# B&R Automation Studio project DemoWall
Automation Studio 4.3.6.57 SP; technology packages: Acp10Arnc0 3.18.2, mapp 1.62.1

## Configuration HardwareConfig1

CPU X20CP1382, AutomationRuntime E4.34, Build 4.1.2, Vc V4.34.3, Safety 1.6

### Task classes (Cpu.sw)
```
Cyclic#1:
  AnalogInpu <- Sources.SimPanel.AnalogInputControl.AnalogInputControl.prg
  DigitalInp <- Sources.SimPanel.DigitalInputControl.DigitalInputControl.prg
  AnalogOutp <- Sources.SimPanel.AnalogOutputControl.AnalogOutputControl.prg
  DigitalOup <- Sources.SimPanel.DigitalOutputControl.DigitalOuputControl.prg
DataObjects: Acp10sys
NcDataObjects: acp10etxen <- DriveAxisConfig.AxisAdditionalFiles.acp10etxen.dob, gAxis01a <- DriveAxisConfig.ACOPOS_P3_3axis.gAxis01obj.gAxis01a.dob, gAxis01i <- DriveAxisConfig.ACOPOS_P3_3axis.gAxis01obj.gAxis01i.dob, gAxis02a <- DriveAxisConfig.ACOPOS_P3_3axis.gAxis02obj.gAxis02a.dob, gAxis02i <- DriveAxisConfig.ACOPOS_P3_3axis.gAxis02obj.gAxis02i.dob, gAxis03a <- DriveAxisConfig.ACOPOS_P3_3axis.gAxis03obj.gAxis03a.dob, gAxis03i <- DriveAxisConfig.ACOPOS_P3_3axis.gAxis03obj.gAxis03i.dob, gAxis04a <- DriveAxisConfig.ACOPOS_micro.gAxis04obj.gAxis04a.dob, gAxis04i <- DriveAxisConfig.ACOPOS_micro.gAxis04obj.gAxis04i.dob, gAxis05a <- DriveAxisConfig.ACOPOS_P3_1axis.gAxis05obj.gAxis05a.dob, gAxis05i <- DriveAxisConfig.ACOPOS_P3_1axis.gAxis05obj.gAxis05i.dob, gAxis06a <- DriveAxisConfig.ACOPOSmicro_stepper.gAxis06obj.gAxis06a.dob, gAxis06i <- DriveAxisConfig.ACOPOSmicro_stepper.gAxis06obj.gAxis06i.dob
Binaries: udbdef, TCData, sysconf, ashwd, ashwac, User, asfw, arconfig, asnxdb1, iomap, Role, Acp10map, acp10cfg
Libraries: Acp10man, Acp10par, NcGlobal, Acp10_MC, brsystem, sys_lib, runtime, Acp10sdc, AsBrStr, OutputLib, asieccon, powerlnk, astime, fileio
```

### Hardware
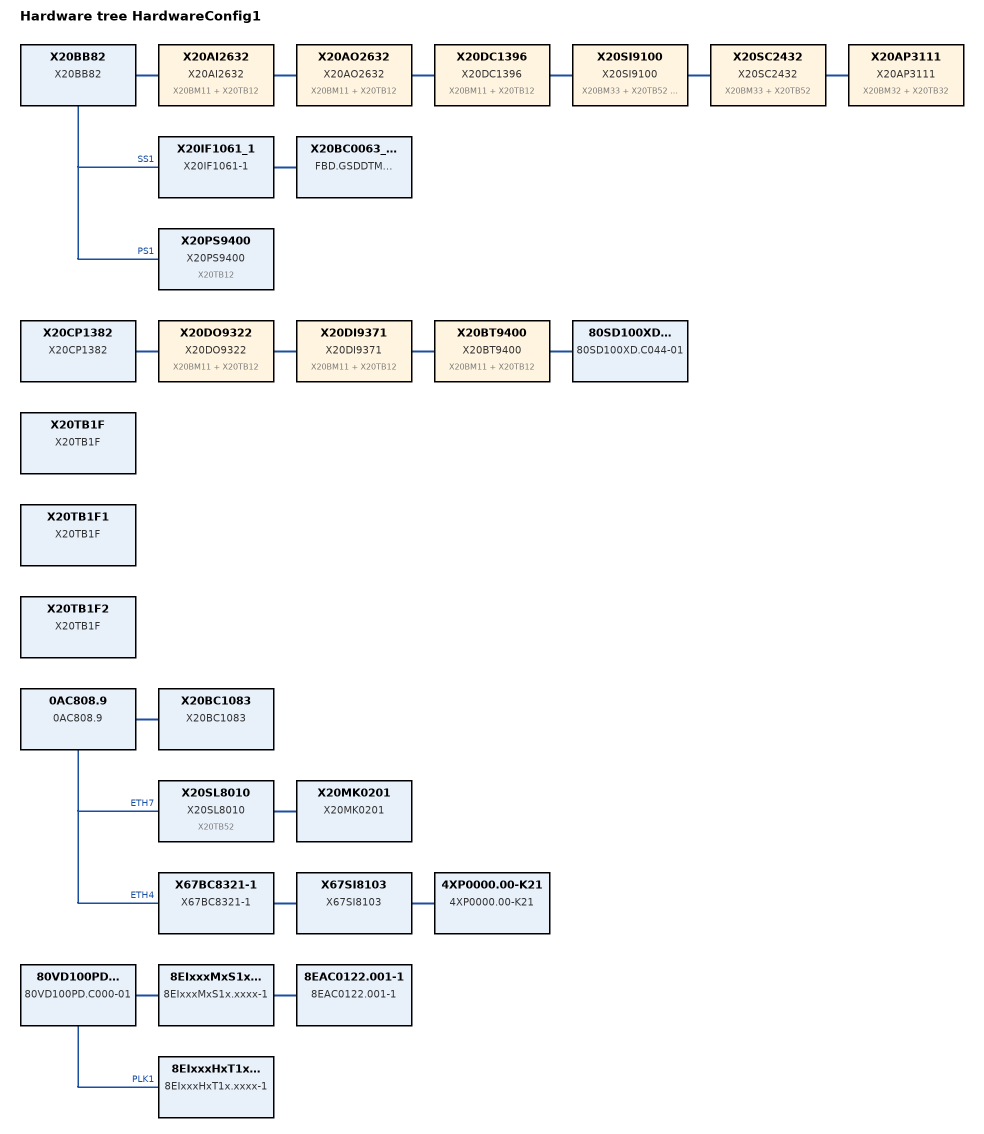
```
0AC808.9 : 0AC808.9 v1.0.0.0  [ETH1 -> 8EIxxxHxT1x.xxxx-1.PLK2 [Cable Type=PowerlinkCable, Length=10, Version=1.0.0.1]; ETH3 -> X20BC1083.PLK1 [Cable Type=PowerlinkCable, Length=10, Version=1.0.0.1]; ETH4 -> X67BC8321-1.PLK1 [Cable Type=PowerlinkCable, Length=10, Version=1.0.0.1]; ETH7 -> X20SL8010.PLK2 [Cable Type=PowerlinkCable, Length=10, Version=1.0.0.1]]
4XP0000.00-K21 : 4XP0000.00-K21 v2.0.0.0  [X2X1 -> X67SI8103.X2X2 [Cable Type=X2XCable, Length=10, Version=1.0.0.1]]
80SD100XD.C044-01 : 80SD100XD.C044-01 v2.1.0.1  [X2X1 -> X20BT9400.X2X1 [Cable Type=X2XCable, Length=10, Version=1.0.0.1]]
  BothEndSwitchesAreNormallyOpen_r1 = on
  QuickStopIsNormallyOpen_r1 = on
80VD100PD.C000-01 : 80VD100PD.C000-01 v2.0.1.0  [PLK1 -> 8EIxxxHxT1x.xxxx-1.PLK1 (NodeNumber=7) [Cable Type=PowerlinkCable, Length=10, Version=1.0.0.1]; PLK2 -> 8EIxxxMxS1x.xxxx-1.PLK1 (NodeNumber=7) [Cable Type=PowerlinkCable, Length=10, Version=1.0.0.1]]
  BothEndSwitchesAreNormallyOpen_r1 = on
  QuickStopIsNormallyOpen_r1 = on
  BothEndSwitchesAreNormallyOpen_r2 = on
  QuickStopIsNormallyOpen_r2 = on
8EAC0122.001-1 : 8EAC0122.001-1 v1.0.0.2  [SS -> 8EIxxxMxS1x.xxxx-1.SS1]
8EIxxxHxT1x.xxxx-1 : 8EIxxxHxT1x.xxxx-1 v1.0.0.3  [PLK1 -> 80VD100PD.C000-01.PLK1 [Cable Type=PowerlinkCable, Length=10, Version=1.0.0.1]; PLK2 -> 0AC808.9.ETH1 [Cable Type=PowerlinkCable, Length=10, Version=1.0.0.1]]
  StandAloneDrive_PowerSupply = dc_powered
  BothEndSwitchesAreNormallyOpen_r1 = on
  QuickStopIsNormallyOpen_r1 = on
  BothEndSwitchesAreNormallyOpen_r2 = on
  QuickStopIsNormallyOpen_r2 = on
  BothEndSwitchesAreNormallyOpen_r3 = on
  QuickStopIsNormallyOpen_r3 = on
8EIxxxMxS1x.xxxx-1 : 8EIxxxMxS1x.xxxx-1 v1.0.0.1  [PLK1 -> 80VD100PD.C000-01.PLK2 [Cable Type=PowerlinkCable, Length=10, Version=1.0.0.1]]
  StandAloneDrive_PowerSupply = dc_powered
  BothEndSwitchesAreNormallyOpen_r1 = on
  QuickStopIsNormallyOpen_r1 = on
X20AI2632 : X20AI2632 v1.1.5.1  [SS1 -> X20TB12d.SS; SL -> X20BM11c.SL1]
X20AO2632 : X20AO2632 v1.0.1.1  [SS1 -> X20TB12e.SS; SL -> X20BM11d.SL1]
X20AP3111 : X20AP3111 v1.0.4.0  [SS1 -> X20TB32.SS; SL -> X20BM32.SL1]
X20BB82 : X20BB82 v1.0.1.0
X20BC0063__DTM_ : FBD.GSDDTM.DTMDev.X20BC0063.1.44 v1.44 (OrderNumber=X20BC0063 (DTM))  [PRB1 -> X20IF1061_1.IF1 (NodeNumber=2)]
  DtmId = 283e3c79-1dfa-4388-8efc-c9f881ac2cf0
  DtmRef = FBD.GSDDTM.DTMDev.X20BC0063.1.44
  ChannelBlocks_f88dcef4-4201-4533-86a5-1206db71a6c6  // X20 DO 9322: 12 DO (24V Source) <Slot 2>
  IO_InputImage_f88dcef4-4201-4533-86a5-1206db71a6c6  // 2 Byte(s)
  IO_OutputImage_f88dcef4-4201-4533-86a5-1206db71a6c6  // 2 Byte(s)
  Channel_1_IO_OutputImage_f88dcef4-4201-4533-86a5-1206db71a6c6
  Name_Channel_1_IO_OutputImage_f88dcef4-4201-4533-86a5-1206db71a6c6 = DigitalOutput01
  Channel_2_IO_OutputImage_f88dcef4-4201-4533-86a5-1206db71a6c6
  Name_Channel_2_IO_OutputImage_f88dcef4-4201-4533-86a5-1206db71a6c6 = DigitalOutput02
  Channel_3_IO_OutputImage_f88dcef4-4201-4533-86a5-1206db71a6c6
  Name_Channel_3_IO_OutputImage_f88dcef4-4201-4533-86a5-1206db71a6c6 = DigitalOutput03
  Channel_4_IO_OutputImage_f88dcef4-4201-4533-86a5-1206db71a6c6
  Name_Channel_4_IO_OutputImage_f88dcef4-4201-4533-86a5-1206db71a6c6 = DigitalOutput04
  Channel_5_IO_OutputImage_f88dcef4-4201-4533-86a5-1206db71a6c6
  Name_Channel_5_IO_OutputImage_f88dcef4-4201-4533-86a5-1206db71a6c6 = DigitalOutput05
  Channel_6_IO_OutputImage_f88dcef4-4201-4533-86a5-1206db71a6c6
  Name_Channel_6_IO_OutputImage_f88dcef4-4201-4533-86a5-1206db71a6c6 = DigitalOutput06
  Channel_7_IO_OutputImage_f88dcef4-4201-4533-86a5-1206db71a6c6
  Name_Channel_7_IO_OutputImage_f88dcef4-4201-4533-86a5-1206db71a6c6 = DigitalOutput07
  Channel_8_IO_OutputImage_f88dcef4-4201-4533-86a5-1206db71a6c6
  Name_Channel_8_IO_OutputImage_f88dcef4-4201-4533-86a5-1206db71a6c6 = DigitalOutput08
X20BC1083 : X20BC1083 v2.5.3.0  [PLK1 -> 0AC808.9.ETH3 [Cable Type=PowerlinkCable, Length=10, Version=1.0.0.1]; PLK2 -> X20CP1382.IF3 [Cable Type=PowerlinkCable, Length=10, Version=1.0.0.1]; SL -> X20BB82.SL1]
X20BM11 : X20BM11 v1.0.0.1  [X2X1 -> X20CP1382.IF6]
X20BM11a : X20BM11 v1.0.0.1  [X2X1 -> X20BM11.X2X2]
X20BM11b : X20BM11 v1.0.0.1  [X2X1 -> X20BM11a.X2X2]
X20BM11c : X20BM11 v1.0.0.1  [X2X1 -> X20BB82.IF1]
X20BM11d : X20BM11 v1.0.0.1  [X2X1 -> X20BM11c.X2X2]
X20BM11e : X20BM11 v1.0.0.1  [X2X1 -> X20BM11d.X2X2]
X20BM32 : X20BM32 v1.0.0.1  [X2X1 -> X20BM33a.X2X2]
X20BM33 : X20BM33 v1.0.0.4  [X2X1 -> X20BM11e.X2X2]
X20BM33a : X20BM33 v1.0.0.4  [X2X1 -> X20BM33.X2X2]
X20BT9400 : X20BT9400 v1.0.2.0  [SS1 -> X20TB12b.SS; SL -> X20BM11b.SL1]
X20CP1382 : X20CP1382 v1.3.2.0  [X1 -> X1.SL; X2 -> X2.SL; X3 -> X3.SL]
  Module X1 (Type=X1, Virtual=true, Version=1.3.2.0)
    Connection (Connector=SS1, TargetModule=X20TB1F, TargetConnector=SS)
    Connection (Connector=SL, TargetModule=X20CP1382, TargetConnector=X1)
  Module X2 (Type=X2, Virtual=true, Version=1.3.2.0)
    Connection (Connector=SS1, TargetModule=X20TB1F1, TargetConnector=SS)
    Connection (Connector=SL, TargetModule=X20CP1382, TargetConnector=X2)
  Module X3 (Type=X3, Virtual=true, Version=1.3.2.0)
    Connection (Connector=SS1, TargetModule=X20TB1F2, TargetConnector=SS)
    Connection (Connector=SL, TargetModule=X20CP1382, TargetConnector=X3)
  Connector IF2:
    ActivateDevice = 1
  ConfigurationID = DemoWall_HardwareConfig1
  Simulation = 1
  TimerDeviceType = EPLX2X
  TimerDevice = X20CP1382.IF3
  Cyclic1Tolerance = 0
  Cyclic1Output = 1
X20DC1396 : X20DC1396 v1.1.0.1  [SS1 -> X20TB12f.SS; SL -> X20BM11e.SL1]
X20DI9371 : X20DI9371 v1.0.2.0  [SS1 -> X20TB12a.SS; SL -> X20BM11a.SL1]
X20DO9322 : X20DO9322 v1.0.3.0  [SS1 -> X20TB12.SS; SL -> X20BM11.SL1]
X20IF1061_1 : X20IF1061-1 v1.6.1.0  [SS -> X20BB82.SS1]
  Connector IF1:
    DtmRef = FBDIF.Hilscher.PBMDtmNX.NETX 100 DP/DPM
    DtmId = 20ba073a-ca99-40f6-b4e4-a2b30d473d5a
  ConfigFile = X20IF1061_1.dtm
  ConfigModule = asnxdb1
X20MK0201 : X20MK0201 v1.0.0.0  [SL -> X20SL8010.SL1]
X20PS9400 : X20PS9400 v1.0.2.4  [SS1 -> X20TB12c.SS; PS -> X20BB82.PS1]
X20SC2432 : X20SC2432 v1.10.0.2  [SS1 -> X20TB52b.SS; SL -> X20BM33a.SL1]
  SafeModuleID = 3
X20SI9100 : X20SI9100 v1.10.0.2  [SS1 -> X20TB52.SS; SS2 -> X20TB52a.SS; SL -> X20BM33.SL1]
X20SL8010 : X20SL8010 v1.6.5.1  [PLK2 -> 0AC808.9.ETH7 [Cable Type=PowerlinkCable, Length=10, Version=1.0.0.1]; SS1 -> X20TB52c.SS]
  SafeProject = SafeLOGIC-1
X20TB12 : X20TB12 v1.0.0.0
X20TB12a : X20TB12 v1.0.0.0
X20TB12b : X20TB12 v1.0.0.0
X20TB12c : X20TB12 v1.0.0.0
X20TB12d : X20TB12 v1.0.0.0
X20TB12e : X20TB12 v1.0.0.0
X20TB12f : X20TB12 v1.0.0.0
X20TB1F : X20TB1F v1.0.0.0
X20TB1F1 : X20TB1F v1.0.0.0
X20TB1F2 : X20TB1F v1.0.0.0
X20TB32 : X20TB32 v1.0.0.1
X20TB52 : X20TB52 v1.0.0.1
X20TB52a : X20TB52 v1.0.0.1
X20TB52b : X20TB52 v1.0.0.1
X20TB52c : X20TB52 v1.0.0.1
X67BC8321-1 : X67BC8321-1 v2.5.3.0  [PLK1 -> 0AC808.9.ETH4 [Cable Type=PowerlinkCable, Length=10, Version=1.0.0.1]]
X67SI8103 : X67SI8103 v1.10.0.1  [X2X1 -> X67BC8321-1.IF1 [Cable Type=X2XCable, Length=10, Version=1.0.0.1]]
  SafeModuleID = 4
```

### IoMap.iom - X20CP1382/IoMap.iom
```iecst
VAR_CONFIG
	Cyclic#1.gAxis05_DrvIf.iLifeCnt AT %IB."80SD100XD.C044-01".LifeCnt;
	Cyclic#1.gAxis05_DrvIf.iDrvOK AT %IX."80SD100XD.C044-01".DrvOk01;
	Cyclic#1.gAxis05_DrvIf.oBoostCurrent AT %QX."80SD100XD.C044-01".BoostCurrent01;
	Cyclic#1.gAxis05_DrvIf.oStandStillCurrent AT %QX."80SD100XD.C044-01".StandstillCurrent01;
	Cyclic#1.gAxis05_DrvIf.oSetTime AT %QW."80SD100XD.C044-01".SetTime01;
	Cyclic#1.gAxis05_MotorStep0 AT %QW."80SD100XD.C044-01".Motor1Step0;
	Cyclic#1.gAxis05_DiDoIf.iLifeCntDriveEnable AT %IB."80SD100XD.C044-01".LifeCnt;
	Cyclic#1.gAxis05_DiDoIf.iLifeCntDriveReady AT %IB."80SD100XD.C044-01".LifeCnt;
	Cyclic#1.gAxis05_DiDoIf.iDriveReady AT %IX."80SD100XD.C044-01".DrvOk01;
	Cyclic#1.gAxis05_DiDoIf.oDriveEnable AT %QX."80SD100XD.C044-01".DriveEnable01;
	Cyclic#1.gAxis05_EncIf1.iLifeCnt AT %IB."80SD100XD.C044-01".LifeCnt;
	Cyclic#1.gAxis05_EncIf1.iEncOK AT %IX."80SD100XD.C044-01".EncOk01;
	Cyclic#1.gAxis05_EncIf1.iActPos AT %IW."80SD100XD.C044-01".ActPos01;
	Cyclic#1.gAxis05_EncIf1.iRefPulsePos AT %IW."80SD100XD.C044-01".RefPulsePos01;
	Cyclic#1.gAxis05_EncIf1.iRefPulseCnt AT %IB."80SD100XD.C044-01".RefPulseCnt01;
	Cyclic#1.gAxis05_EncIf1.iActTime AT %IW."80SD100XD.C044-01".ActTime01;
	::gdiSim1 AT %IX."X20DI9371".DigitalInput01;
	::gdiSim2 AT %IX."X20DI9371".DigitalInput02;
	::gdiSim3 AT %IX."X20DI9371".DigitalInput03;
	::gdiSim4 AT %IX."X20DI9371".DigitalInput04;
	::gdiSim5 AT %IX."X20DI9371".DigitalInput05;
	::gdiSim6 AT %IX."X20DI9371".DigitalInput06;
	::gdiSim7 AT %IX."X20DI9371".DigitalInput07;
	::gdiSim8 AT %IX."X20DI9371".DigitalInput08;
	::gdoSim1 AT %QX."X20DO9322".DigitalOutput01;
	::gdoSim2 AT %QX."X20DO9322".DigitalOutput02;
	::gdoSim3 AT %QX."X20DO9322".DigitalOutput03;
	::gdoSim4 AT %QX."X20DO9322".DigitalOutput04;
	::gdoSim5 AT %QX."X20DO9322".DigitalOutput05;
	::gdoSim6 AT %QX."X20DO9322".DigitalOutput06;
	::gdoSim7 AT %QX."X20DO9322".DigitalOutput07;
	::gdoSim8 AT %QX."X20DO9322".DigitalOutput08;
	::gaiSim1 AT %IW."X20AI2632".AnalogInput01;
	::gaiSim2 AT %IW."X20AI2632".AnalogInput02;
	::gaoSim1 AT %QW."X20AO2632".AnalogOutput01;
	::gaoSim2 AT %QW."X20AO2632".AnalogOutput02;
END_VAR
```

### Acp10cfg.ncc - X20CP1382/Motion/Acp10cfg.ncc
```
NcConfiguration (Version=3.18.2, NcSwId=Acp10)
  ACP10CF1_typ:
    cnt_nettrc_rec_drive = 1500
    bufsize_trace_upload = 1200
    tc_nc_man_task = Cyclic #1
    glob_pv_as_ncobject = Yes
    ncsys_dl_broadcast = Yes
    ncsys_dl_acp_reset = Yes
    safemc_log_err_to_ax = Yes
    network_init:
      ncsw_init_execute = Yes
      automatic_execute = No
      node_nr_warning = Yes
      net_err_before_ncact = Yes
    nettrc:
      enter_parsecrec = Yes
      enter_ncaction = Yes
      save_ring_startidx = Yes
    cam_prof_download:
      cam_dat_dl_parallel = No
      tc_cam_dl_parallel = Task class for NC Manager task
    plk_if[0]:
      if_name = IF3
      tc_CycDat_PLCopen = Task class for NC Manager task
      mc_broadcast_extdat = No
    sdc_if[0]:
      if_name = SDC_IF1
      mc_broadcast_size = 800
      mc_broadcast_extdat = No
```

### Acp10map.ncm - X20CP1382/Motion/Acp10map.ncm
```
NcMapping (NcSwId=Acp10)
  NcObject gAxis01 (ModuleId=8EIxxxHxT1x.xxxx-1, Type=ncAXIS, Channel=1, AcoposSimulation=Off, InitParameter=gAxis01i, AcoposParameter=gAxis01a, Disabled=FALSE, ModuleDisabled=FALSE)
  NcObject gAxis02 (ModuleId=8EIxxxHxT1x.xxxx-1, Type=ncAXIS, Channel=2, AcoposSimulation=Off, InitParameter=gAxis02i, AcoposParameter=gAxis02a, Disabled=FALSE, ModuleDisabled=FALSE)
  NcObject gAxis03 (ModuleId=8EIxxxHxT1x.xxxx-1, Type=ncAXIS, Channel=3, AcoposSimulation=Off, InitParameter=gAxis03i, AcoposParameter=gAxis03a, Disabled=FALSE, ModuleDisabled=FALSE)
  NcObject 8EIxxxHxT1x.xxxx-1_ncV_AXIS1 (ModuleId=8EIxxxHxT1x.xxxx-1, Type=ncV_AXIS, Channel=1, Disabled=TRUE, ModuleDisabled=FALSE)
  NcObject 8EIxxxHxT1x.xxxx-1_ncV_AXIS2 (ModuleId=8EIxxxHxT1x.xxxx-1, Type=ncV_AXIS, Channel=2, Disabled=TRUE, ModuleDisabled=FALSE)
  NcObject 8EIxxxHxT1x.xxxx-1_ncV_AXIS3 (ModuleId=8EIxxxHxT1x.xxxx-1, Type=ncV_AXIS, Channel=3, Disabled=TRUE, ModuleDisabled=FALSE)
  NcObject gAxis04 (ModuleId=80VD100PD.C000-01, Type=ncAXIS, Channel=1, AcoposSimulation=Off, InitParameter=gAxis04i, AcoposParameter=gAxis04a, Disabled=FALSE, ModuleDisabled=FALSE)
  NcObject 80VD100PD.C000-01_ncAXIS2 (ModuleId=80VD100PD.C000-01, Type=ncAXIS, Channel=2, AcoposSimulation=Off, Disabled=TRUE, ModuleDisabled=FALSE)
  NcObject 80VD100PD.C000-01_ncV_AXIS1 (ModuleId=80VD100PD.C000-01, Type=ncV_AXIS, Channel=1, Disabled=TRUE, ModuleDisabled=FALSE)
  NcObject 80VD100PD.C000-01_ncV_AXIS2 (ModuleId=80VD100PD.C000-01, Type=ncV_AXIS, Channel=2, Disabled=TRUE, ModuleDisabled=FALSE)
  NcObject gAxis05 (ModuleId=80SD100XD.C044-01, ModuleAddress=SDC_IF1.ST1, Type=ncAXIS, Channel=1, AcoposSimulation=Off, InitParameter=gAxis05i, AcoposParameter=gAxis05a, Disabled=FALSE, ModuleDisabled=FALSE)
  NcObject 80SD100XD.C044-01_ncAXIS2 (ModuleId=80SD100XD.C044-01, ModuleAddress=SDC_IF1.ST2, Type=ncAXIS, Channel=1, AcoposSimulation=Off, Disabled=TRUE, ModuleDisabled=FALSE)
  NcObject gAxis06 (ModuleId=8EIxxxMxS1x.xxxx-1, Type=ncAXIS, Channel=1, AcoposSimulation=Off, InitParameter=gAxis06i, AcoposParameter=gAxis06a, Disabled=FALSE, ModuleDisabled=FALSE)
  NcObject 8EIxxxMxS1x.xxxx-1_ncV_AXIS1 (ModuleId=8EIxxxMxS1x.xxxx-1, Type=ncV_AXIS, Channel=1, Disabled=TRUE, ModuleDisabled=FALSE)
```

## Logical view

Binary libraries used (declarations not repeated): operator, runtime, astime, AsIecCon, Acp10man 3.18.2, Acp10par 3.18.2, NcGlobal 3.18.2, Acp10_MC 3.18.2, brsystem, sys_lib, Acp10sdc 3.18.2, AsBrStr

### Package Logical/Libraries - Global libraries

### gInputOutput.var
```iecst
VAR
	gdiSim1 : BOOL := FALSE; (*4sim.00-01 *)
	gdiSim2 : BOOL := FALSE; (*4sim.00-01 *)
	gdiSim3 : BOOL := FALSE; (*4sim.00-01 *)
	gdiSim4 : BOOL := FALSE; (*4sim.00-01 *)
	gdiSim5 : BOOL := FALSE; (*4sim.00-01 *)
	gdiSim6 : BOOL := FALSE; (*4sim.00-01 *)
	gdiSim7 : BOOL := FALSE; (*4sim.00-01 *)
	gdiSim8 : BOOL := FALSE; (*4sim.00-01 *)
	gdoSim1 : BOOL := FALSE; (*4sim.00-01 *)
	gdoSim2 : BOOL := FALSE; (*4sim.00-01 *)
	gdoSim3 : BOOL := FALSE; (*4sim.00-01 *)
	gdoSim4 : BOOL := FALSE; (*4sim.00-01 *)
	gdoSim5 : BOOL := FALSE; (*4sim.00-01 *)
	gdoSim6 : BOOL := FALSE; (*4sim.00-01 *)
	gdoSim7 : BOOL := FALSE; (*4sim.00-01 *)
	gdoSim8 : BOOL := FALSE; (*4sim.00-01 *)
	gaiSim1 : INT; (*4sim.00-01 *)
	gaiSim2 : INT; (*4sim.00-01 *)
	gaoSim1 : INT; (*4sim.00-01 *)
	gaoSim2 : INT; (*4sim.00-01 *)
	gdcSim1 : USINT; (*4sim.00-01  digital counter*)
END_VAR
```

### Program Logical/Sources/SimPanel/DigitalInputControl/DigitalInputControl (IEC)

#### DigitalInputControl.st - Init, cyclic, exit code
```iecst
PROGRAM _INIT

END_PROGRAM

PROGRAM _CYCLIC

	DigitalInput1.Status := gdiSim1;
	DigitalInput2.Status := gdiSim2;
	DigitalInput3.Status := gdiSim3;
	DigitalInput4.Status := gdiSim4;
	DigitalInput5.Status := gdiSim5;
	DigitalInput6.Status := gdiSim6;
	DigitalInput7.Status := gdiSim7;
	DigitalInput8.Status := gdiSim8;

END_PROGRAM

PROGRAM _EXIT

END_PROGRAM
```

#### DigitalInput.typ
```iecst
TYPE
	DigitalInputType : 	STRUCT
		Status : BOOL;
	END_STRUCT;
END_TYPE
```

#### DigitalInput.var - Local variables
```iecst
VAR
	DigitalInput1 : DigitalInputType;
	DigitalInput2 : DigitalInputType;
	DigitalInput3 : DigitalInputType;
	DigitalInput4 : DigitalInputType;
	DigitalInput5 : DigitalInputType;
	DigitalInput6 : DigitalInputType;
	DigitalInput7 : DigitalInputType;
	DigitalInput8 : DigitalInputType;
END_VAR
```

### Library Logical/Sources/SimPanel/DigitalOutputControl/OutputLib (IEC)

#### OutputLib.fun - Exported functions and function blocks
```iecst
{REDUND_OK} FUNCTION DigitalOutputFunction : BOOL (*Obsługa Digital Outputa z opcUA*) (*$GROUP=User,$CAT=User,$GROUPICON=User.png,$CATICON=User.png*)
	VAR_IN_OUT
		On : BOOL;
		Off : BOOL;
		Status : BOOL;
	END_VAR
END_FUNCTION
```

#### DigitalOutputFunction.st
```iecst
(* Obsługa Digital Outputa z opcUA *)
FUNCTION DigitalOutputFunction

	IF Off THEN
		Off := 0;
		Status := 0;
	END_IF;

	IF On THEN
		On := 0 ;
		Status := 1;
	END_IF;

END_FUNCTION
```

### Program Logical/Sources/SimPanel/DigitalOutputControl/DigitalOuputControl (IEC)

#### DigitalOuputControl.st - Init, cyclic, exit code
```iecst
PROGRAM _INIT

END_PROGRAM

PROGRAM _CYCLIC

	DigitalOutputFunction(DigitalOutput1.Commands.On, DigitalOutput1.Commands.Off, DigitalOutput1.Status);
	DigitalOutputFunction(DigitalOutput2.Commands.On, DigitalOutput2.Commands.Off, DigitalOutput2.Status);
	DigitalOutputFunction(DigitalOutput3.Commands.On, DigitalOutput3.Commands.Off, DigitalOutput3.Status);
	DigitalOutputFunction(DigitalOutput4.Commands.On, DigitalOutput4.Commands.Off, DigitalOutput4.Status);
	DigitalOutputFunction(DigitalOutput5.Commands.On, DigitalOutput5.Commands.Off, DigitalOutput5.Status);
	DigitalOutputFunction(DigitalOutput6.Commands.On, DigitalOutput6.Commands.Off, DigitalOutput6.Status);
	DigitalOutputFunction(DigitalOutput7.Commands.On, DigitalOutput7.Commands.Off, DigitalOutput7.Status);
	DigitalOutputFunction(DigitalOutput8.Commands.On, DigitalOutput8.Commands.Off, DigitalOutput8.Status);

	gdoSim1 := DigitalOutput1.Status;
	gdoSim2 := DigitalOutput2.Status;
	gdoSim3 := DigitalOutput3.Status;
	gdoSim4 := DigitalOutput4.Status;
	gdoSim5 := DigitalOutput5.Status;
	gdoSim6 := DigitalOutput6.Status;
	gdoSim7 := DigitalOutput7.Status;
	gdoSim8 := DigitalOutput8.Status;

END_PROGRAM

PROGRAM _EXIT

END_PROGRAM
```

#### DitgitalOutput.typ
```iecst
TYPE
	DigitalOutputType : 	STRUCT
		Status : BOOL;
		Commands : CommandType;
	END_STRUCT;
	CommandType : 	STRUCT
		On : BOOL;
		Off : BOOL;
	END_STRUCT;
END_TYPE
```

#### DigitalOutput.var - Local variables
```iecst
VAR
	DigitalOutput1 : DigitalOutputType;
	DigitalOutput2 : DigitalOutputType;
	DigitalOutput3 : DigitalOutputType;
	DigitalOutput4 : DigitalOutputType;
	DigitalOutput5 : DigitalOutputType;
	DigitalOutput6 : DigitalOutputType;
	DigitalOutput7 : DigitalOutputType;
	DigitalOutput8 : DigitalOutputType;
END_VAR
```

### gAnalogInput.typ
```iecst
TYPE
	gAnalogInputType : 	STRUCT
		BaseValue : INT;
		ScaledValue : REAL;
	END_STRUCT;
END_TYPE
```

### gAnalogInput.var - Local variables
```iecst
VAR
	gAnalogInput1 : gAnalogInputType;
	gAnalogInput2 : gAnalogInputType;
END_VAR
```

### Program Logical/Sources/SimPanel/AnalogInputControl/AnalogInputControl (IEC)

#### AnalogInputControl.st - Init, cyclic, exit code
```iecst
PROGRAM _INIT

END_PROGRAM

PROGRAM _CYCLIC

	gAnalogInput1.BaseValue := gaiSim1;
	gAnalogInput2.BaseValue := gaiSim2;

	gAnalogInput1.ScaledValue := (gAnalogInput1.BaseValue/32767.0)*9.8;
	gAnalogInput2.ScaledValue := (gAnalogInput2.BaseValue/32767.0)*9.8;

END_PROGRAM

PROGRAM _EXIT

END_PROGRAM
```

### gAnalogOutput.var - Local variables
```iecst
VAR
	gAnalogOutput1 : gAnalogOutputType;
	gAnalogOutput2 : gAnalogOutputType;
END_VAR
```

### gAnalogOuput.typ
```iecst
TYPE
	gAnalogOutputType : 	STRUCT
		BaseValue : REAL;
		ScaledValue : INT;
	END_STRUCT;
END_TYPE
```

### Program Logical/Sources/SimPanel/AnalogOutputControl/AnalogOutputControl (IEC)

#### AnalogOutputControl.st - Init, cyclic, exit code
```iecst
PROGRAM _INIT

END_PROGRAM

PROGRAM _CYCLIC

	gAnalogOutput1.ScaledValue := REAL_TO_INT(gAnalogOutput1.BaseValue * 32676.0 / 9.8);
	gAnalogOutput2.ScaledValue := REAL_TO_INT(gAnalogOutput2.BaseValue * 32676.0 / 9.8);

	gaoSim1 := gAnalogOutput1.ScaledValue;
	gaoSim2 := gAnalogOutput2.ScaledValue;

END_PROGRAM

PROGRAM _EXIT

END_PROGRAM
```

### gAxisStructures.var - Global variables
```iecst
VAR
	gAxis01 : ACP10AXIS_typ;
	gAxis02 : ACP10AXIS_typ;
	gAxis03 : ACP10AXIS_typ;
	gAxis04 : ACP10AXIS_typ;
	gAxis05 : ACP10AXIS_typ;
	gAxis05_HW : SdcHwCfg_typ := (0);
	gAxis05_DrvIf : SdcDrvIf16_typ := (0);
	gAxis05_EncIf1 : SdcEncIf16_typ := (0);
	gAxis05_DiDoIf : SdcDiDoIf_typ := (0);
	gAxis05_MotorStep0 : INT := 0;
	gAxis06 : ACP10AXIS_typ;
END_VAR
```


- Data object Logical/DriveAxisConfig/ACOPOS_P3_3axis/gAxis01obj/gAxis01a (Apt) (no source held here)

- Data object Logical/DriveAxisConfig/ACOPOS_P3_3axis/gAxis01obj/gAxis01i (Ax) (no source held here)

- Data object Logical/DriveAxisConfig/ACOPOS_P3_3axis/gAxis02obj/gAxis02a (Apt) (no source held here)

- Data object Logical/DriveAxisConfig/ACOPOS_P3_3axis/gAxis02obj/gAxis02i (Ax) (no source held here)

### Package Logical/DriveAxisConfig/ACOPOS_P3_3axis/gAxis03obj - gAxis03obj

- Data object Logical/DriveAxisConfig/ACOPOS_P3_3axis/gAxis03obj/gAxis03a (Apt) (no source held here)

### Data object Logical/DriveAxisConfig/ACOPOS_P3_3axis/gAxis03obj/gAxis03i (Ax)

#### gAxis03i.ax
```
InitParameter (Version=3.18.2, NcSwId=Acp10)
  ACP10AXIS_typ:
    dig_in:
      level:
        reference = ncACTIV_HI
        pos_hw_end = ncACTIV_HI
        neg_hw_end = ncACTIV_HI
        trigger1 = ncACTIV_HI
        trigger2 = ncACTIV_HI
    encoder_if:
      parameter:
        count_dir = ncSTANDARD
        scaling:
          load:
            units = 1000
            rev_motor = 1
    limit:
      parameter:
        v_pos = 10000
        v_neg = 10000
        a1_pos = 50000
        a2_pos = 50000
        a1_neg = 50000
        a2_neg = 50000
        t_jolt = 0
        t_in_pos = 0
        pos_sw_end = 2000000000
        neg_sw_end = -2000000000
        ds_warning = 500
        ds_stop = 1000
        a_stop = 1.0e30
        dv_stop = 0
        dv_stop_mode = ncOFF
    controller:
      mode = ncPOSITION
      position:
        kv = 50
        tn = 0
        t_predict = 0.0004
        t_total = 0.0004
        p_max = 1.0e30
        i_max = 0
      speed:
        kv = 2.0
        tn = 0
        t_filter = 0.0
        isq_filter1:
          type = ncOFF
          a0 = 0.0
          a1 = 0.0
          b0 = 0.0
          b1 = 0.0
          b2 = 0.0
          c0_par_id = 0
          c1_par_id = 0
        isq_filter2:
          type = ncOFF
          a0 = 0.0
          a1 = 0.0
          b0 = 0.0
          b1 = 0.0
          b2 = 0.0
          c0_par_id = 0
          c1_par_id = 0
        isq_filter3:
          type = ncOFF
          a0 = 0.0
          a1 = 0.0
          b0 = 0.0
          b1 = 0.0
          b2 = 0.0
          c0_par_id = 0
          c1_par_id = 0
      uf:
        type = ncLINEAR
        auto_config = ncMOTOR_PAR
        u0 = 0
        un = 0
        fn = 50.0
        k_f_slip = 0
      ff:
        torque_load = 0.0
        torque_pos = 0.0
        torque_neg = 0.0
        kv_torque = 0.0
        inertia = 0.0
        t_filter_a = 0.0
    move:
      stop:
        parameter[0]:
          decel_ramp = ncA_LIMIT
          controller = ncON
        parameter[1]:
          decel_ramp = ncA_LIMIT
          controller = ncON
        parameter[2]:
          decel_ramp = ncA_LIMIT
          controller = ncON
        parameter[3]:
          decel_ramp = ncA_LIMIT
          controller = ncON
        quickstop:
          decel_ramp = ncA_LIMIT
        drive_error:
          decel_ramp = ncA_LIMIT
      homing:
        parameter:
          s = 0
          v_switch = 5000
          v_trigger = 500
          a = 50000
          mode = ncDIRECT
          edge_sw = ncPOSITIVE
          start_dir = ncPOSITIVE
          trigg_dir = ncPOSITIVE
          ref_pulse = ncOFF
          fix_dir = ncOFF
          tr_s_block = 0
          torque_lim = 0
          ds_block = 0
          ds_stop = 0
      basis:
        parameter:
          v_pos = 5000
          v_neg = 5000
          a1_pos = 50000
          a2_pos = 50000
          a1_neg = 50000
          a2_neg = 50000
    message:
      text:
        parameter:
          format = ncBREAK
          columns = 80
          data_modul = acp10etxen
```

### Package Logical/DriveAxisConfig/ACOPOS_P3_1axis/gAxis05obj - gAxis05obj

- Data object Logical/DriveAxisConfig/ACOPOS_P3_1axis/gAxis05obj/gAxis05a (Apt) (no source held here)

### Data object Logical/DriveAxisConfig/ACOPOS_P3_1axis/gAxis05obj/gAxis05i (Ax)

#### gAxis05i.ax
```
InitParameter (Version=3.18.2, NcSwId=Acp10)
  ACP10AXIS_typ:
    dig_in:
      level:
        reference = ncACTIV_HI
        pos_hw_end = ncACTIV_HI
        neg_hw_end = ncACTIV_HI
        trigger1 = ncACTIV_HI
        trigger2 = ncACTIV_HI
    encoder_if:
      parameter:
        count_dir = ncSTANDARD
        scaling:
          load:
            units = 1000
            rev_motor = 1
    limit:
      parameter:
        v_pos = 10000
        v_neg = 10000
        a1_pos = 50000
        a2_pos = 50000
        a1_neg = 50000
        a2_neg = 50000
        t_jolt = 0
        t_in_pos = 0
        pos_sw_end = 2000000000
        neg_sw_end = -2000000000
        ds_warning = 500
        ds_stop = 1000
        a_stop = 1.0e30
        dv_stop = 0
        dv_stop_mode = ncOFF
    controller:
      mode = ncPOSITION
      position:
        kv = 50
        tn = 0
        t_predict = 0.01
        t_total = 0.01
        p_max = 1.0e30
        i_max = 0
      speed:
        kv = 2.0
        tn = 0
        t_filter = 0.0
        isq_filter1:
          type = ncOFF
          a0 = 0.0
          a1 = 0.0
          b0 = 0.0
          b1 = 0.0
          b2 = 0.0
          c0_par_id = 0
          c1_par_id = 0
        isq_filter2:
          type = ncOFF
          a0 = 0.0
          a1 = 0.0
          b0 = 0.0
          b1 = 0.0
          b2 = 0.0
          c0_par_id = 0
          c1_par_id = 0
        isq_filter3:
          type = ncOFF
          a0 = 0.0
          a1 = 0.0
          b0 = 0.0
          b1 = 0.0
          b2 = 0.0
          c0_par_id = 0
          c1_par_id = 0
      uf:
        type = ncLINEAR
        auto_config = ncMOTOR_PAR
        u0 = 0
        un = 0
        fn = 50.0
        k_f_slip = 0
      ff:
        torque_load = 0.0
        torque_pos = 0.0
        torque_neg = 0.0
        kv_torque = 0.0
        inertia = 0.0
        t_filter_a = 0.0
    move:
      stop:
        parameter[0]:
          decel_ramp = ncA_LIMIT
          controller = ncON
        parameter[1]:
          decel_ramp = ncA_LIMIT
          controller = ncON
        parameter[2]:
          decel_ramp = ncA_LIMIT
          controller = ncON
        parameter[3]:
          decel_ramp = ncA_LIMIT
          controller = ncON
        quickstop:
          decel_ramp = ncA_LIMIT
        drive_error:
          decel_ramp = ncA_LIMIT
      homing:
        parameter:
          s = 0
          v_switch = 5000
          v_trigger = 500
          a = 50000
          mode = ncDIRECT
          edge_sw = ncPOSITIVE
          start_dir = ncPOSITIVE
          trigg_dir = ncPOSITIVE
          ref_pulse = ncOFF
          fix_dir = ncOFF
          tr_s_block = 0
          torque_lim = 0
          ds_block = 0
          ds_stop = 0
      basis:
        parameter:
          v_pos = 5000
          v_neg = 5000
          a1_pos = 50000
          a2_pos = 50000
          a1_neg = 50000
          a2_neg = 50000
    message:
      text:
        parameter:
          format = ncBREAK
          columns = 80
          data_modul = acp10etxen
```


- Data object Logical/DriveAxisConfig/ACOPOS_micro/gAxis04obj/gAxis04a (Apt) (no source held here)

- Data object Logical/DriveAxisConfig/ACOPOS_micro/gAxis04obj/gAxis04i (Ax) (no source held here)

- Data object Logical/DriveAxisConfig/ACOPOSmicro_stepper/gAxis06obj/gAxis06a (Apt) (no source held here)

- Data object Logical/DriveAxisConfig/ACOPOSmicro_stepper/gAxis06obj/gAxis06i (Ax) (no source held here)

### Program Logical/DriveAxisConfig/AxisAdditionalFiles/ncsdcctrl (IEC)

#### ncsdcctrlCyclic.st
```iecst
PROGRAM _CYCLIC

(* ### BEGIN gAxis05 ### *)

(* life counter emulation of digital inputs *)
       gAxis05_DiDoIf.iLifeCntReference := gAxis05_DiDoIf.iLifeCntReference + 1;
       gAxis05_DiDoIf.iLifeCntNegHwEnd  := gAxis05_DiDoIf.iLifeCntNegHwEnd  + 1;
       gAxis05_DiDoIf.iLifeCntPosHwEnd  := gAxis05_DiDoIf.iLifeCntPosHwEnd  + 1;

(* default function model of ACOPOSmicro: convert absolute steps to delta steps - overflow save delta calculation *)
       gAxis05_MotorStep0 := gAxis05_DrvIf.oSetPos - gAxis05_oSetPosOld;
       gAxis05_oSetPosOld := gAxis05_DrvIf.oSetPos;

(* ### END gAxis05 ### *)

END_PROGRAM
```

#### ncsdcctrlInit.st
```iecst
PROGRAM _INIT

(* ### BEGIN gAxis05 ### *)

(* initialize general interfaces *)
       gAxis05.size := gAxis05.size;
       gAxis05_HW.DrvIf_Typ := ncSDC_DRVSM16;
       brsstrcpy( ADR(gAxis05_HW.DrvIf_Name[0]), ADR('gAxis05_DrvIf') );
       gAxis05_HW.DiDoIf_Typ := ncSDC_DIDO;
       brsstrcpy( ADR(gAxis05_HW.DiDoIf_Name[0]), ADR('gAxis05_DiDoIf') );
       gAxis05_HW.EncIf1_Typ := ncSDC_ENC16;
       brsstrcpy( ADR(gAxis05_HW.EncIf1_Name[0]), ADR('gAxis05_EncIf1') );
       gAxis05_EncIf1.iLifeCnt := gAxis05_EncIf1.iLifeCnt;

(* initialize old-value for delta step calculation *)
       gAxis05_oSetPosOld := gAxis05_DrvIf.oSetPos;

(* ### END gAxis05 ### *)

END_PROGRAM
```

### Data object Logical/DriveAxisConfig/AxisAdditionalFiles/acp10etxen (Ett)

- acp10etxen.ett (not shown)

Listed in the project but not available here: Logical/Sources/SimPanel/DigitalCounterControl, Logical/Sources/DriveControl/DriveAcoposMicro, Logical/Sources/DriveControl/DriveAcoposStepper, Logical/DriveAxisConfig/AxisAdditionalFiles/ncsdcctrl/ncsdcctrl.typ, Logical/DriveAxisConfig/AxisAdditionalFiles/ncsdcctrl/ncsdcctrl.var
